FUNCTION_BLOCK VAV_PRE (* Variable Air Valve Model pre-calculation *)
  (* Standard: 61499-1; Classification: Simulation; ApplicationDomain: HVAC; Function: VAV *)
  (* Version 0.0, 2006-04-10, JHC, Holobloc Inc *)
  (* Compiler header: package fb.rt.hvac; *)
  (* Compiler Java Sun JDK 1.5.0 *)
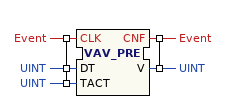
  EVENT_INPUT
    CLK WITH DT, TACT; (* Simulation clock *)
  END_EVENT
  EVENT_OUTPUT
    CNF WITH V; (* Pre-calc complete *)
  END_EVENT
  VAR_INPUT
    DT : UINT := 10; (* CLK period, sec *)
    TACT : UINT := 95; (* Damper actuation time, sec *)
  END_VAR
  VAR_OUTPUT
    V : UINT; (* Open/Close Speed, % per CLK cycle *)
  END_VAR
  ALGORITHM CLK IN Java: (* VAV model pre-calculation *)
V.value = DT.value*100/TACT.value;
if(DT.value>0) V.value = Math.max(V.value,1);
CNF.serviceEvent(this);
  END_ALGORITHM
END_FUNCTION_BLOCK
